(*
Sets the beam class assertion lines for a given beam class.
*)
FUNCTION_BLOCK FB_BeamClassOutputs
VAR_INPUT
    i_ArbiterBP    :    ST_BeamParams;
END_VAR
VAR_OUTPUT
END_VAR
VAR
    wBeamClass    :    BYTE;

    InitCounter: INT;
    counter    :    INT;
    
            {attribute 'TcLinkTo' := '[1] := TIIB[PMPS_BC]^Channel 1^Output;
                              [2] := TIIB[PMPS_BC]^Channel 2^Output;
                              [3] := TIIB[PMPS_BC]^Channel 3^Output;
                              [4] := TIIB[PMPS_BC]^Channel 4^Output;
                              
                              [5] := TIIB[PMPS_BC]^Channel 5^Output;
                              [6] := TIIB[PMPS_BC]^Channel 6^Output;
                              [7] := TIIB[PMPS_BC]^Channel 7^Output;
                              [8] := TIIB[PMPS_BC]^Channel 8^Output;
                              
                              [9] := TIIB[PMPS_BC]^Channel 9^Output;
                              [10] := TIIB[PMPS_BC]^Channel 10^Output;
                              [11] := TIIB[PMPS_BC]^Channel 11^Output;
                              [12] := TIIB[PMPS_BC]^Channel 12^Output;
                              
                              [13] := TIIB[PMPS_BC]^Channel 13^Output;
                              [14] := TIIB[PMPS_BC]^Channel 14^Output;
                              [15] := TIIB[PMPS_BC]^Channel 15^Output;
                              [16] := TIIB[PMPS_BC]^Channel 16^Output'}
    q_BC_ASSERTION_LINES    AT    %Q*    : ARRAY [1..16] OF    BOOL;
END_VAR


//Beam Class
////////////////////////////////////
//0x0 = 0000 0000 0000 0000
//0x1 = 0000 0000 0000 0001
//0xF = 1111 1111 1111 1111

//Initialize BC lines to zero on every pass
FOR InitCounter := 1 TO 16 DO
    q_BC_ASSERTION_LINES[InitCounter] := FALSE;
END_FOR

//Set BC lines according to beam class
//A BC of 0x0 would pass over this loop, setting none of the lines high
// , as FOR loops check the initialized variable at the top to see if it's >
// than the "TO" variable.
FOR wBeamClass:=1 TO i_ArbiterBP.nBeamClass DO
    q_BC_ASSERTION_LINES[wBeamClass] := TRUE;
END_FOR

END_FUNCTION_BLOCK

(* stored: Version 1.1.0.1, ProductVersion 3.1.4022.18
   POU FB_BeamClassOutputs: Id {4a29fded-500d-49a8-af9c-1a0c32a74d5a}, SpecialFunc None *)
